// Mitsubishi GX Works2 project: IOCHECK   PLC: Q03UD

PROGRAM MAIN
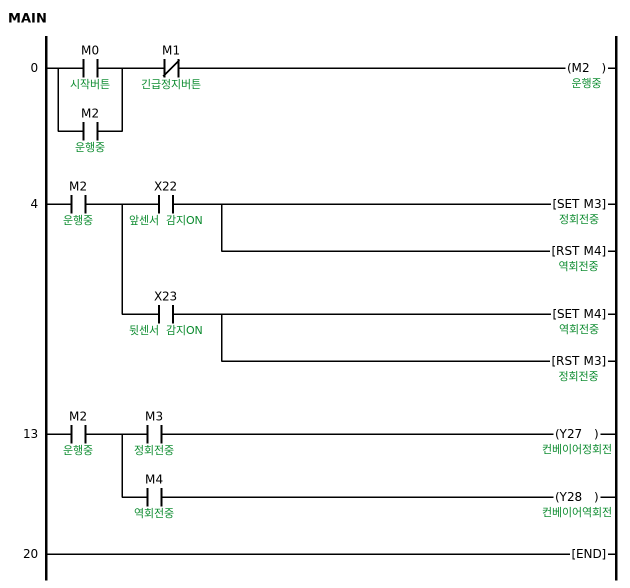
0     LD      M0  ; 시작버튼
      OR      M2  ; 운행중
      ANI     M1  ; 긴급정지버튼
      OUT     M2  ; 운행중
4     LD      M2  ; 운행중
      MPS
      AND     X22  ; 앞센서  감지ON
      SET     M3  ; 정회전중
      RST     M4  ; 역회전중
      MPP
      AND     X23  ; 뒷센서  감지ON
      SET     M4  ; 역회전중
      RST     M3  ; 정회전중
13    LD      M2  ; 운행중
      MPS
      AND     M3  ; 정회전중
      OUT     Y27  ; 컨베이어정회전
      MPP
      AND     M4  ; 역회전중
      OUT     Y28  ; 컨베이어역회전
20    END
END_PROGRAM

PROGRAM IOCHECK
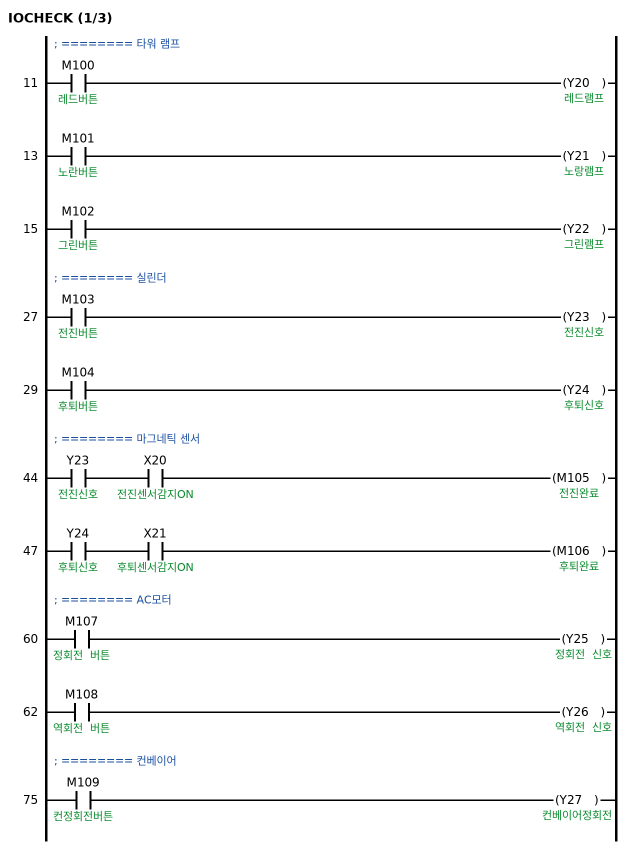
; ======== 타워 램프
11    LD      M100  ; 레드버튼
      OUT     Y20  ; 레드램프
13    LD      M101  ; 노란버튼
      OUT     Y21  ; 노랑램프
15    LD      M102  ; 그린버튼
      OUT     Y22  ; 그린램프
; ======== 실린더
27    LD      M103  ; 전진버튼
      OUT     Y23  ; 전진신호
29    LD      M104  ; 후퇴버튼
      OUT     Y24  ; 후퇴신호
; ======== 마그네틱 센서
44    LD      Y23  ; 전진신호
      AND     X20  ; 전진센서감지ON
      OUT     M105  ; 전진완료
47    LD      Y24  ; 후퇴신호
      AND     X21  ; 후퇴센서감지ON
      OUT     M106  ; 후퇴완료
; ======== AC모터
60    LD      M107  ; 정회전  버튼
      OUT     Y25  ; 정회전  신호
62    LD      M108  ; 역회전  버튼
      OUT     Y26  ; 역회전  신호
; ======== 컨베이어
75    LD      M109  ; 컨정회전버튼
      OUT     Y27  ; 컨베이어정회전
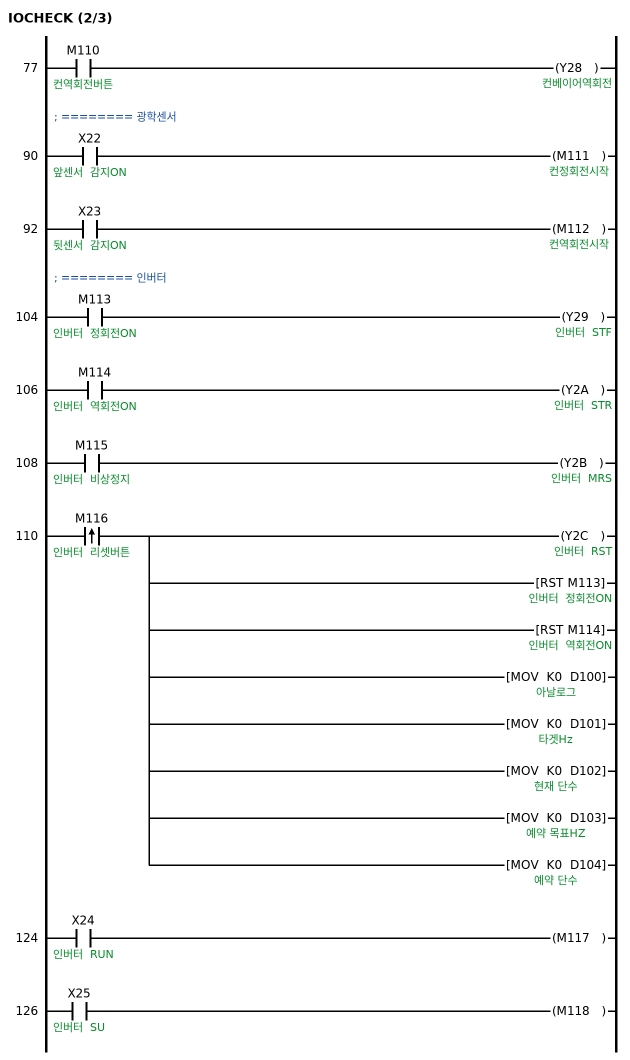
77    LD      M110  ; 컨역회전버튼
      OUT     Y28  ; 컨베이어역회전
; ======== 광학센서
90    LD      X22  ; 앞센서  감지ON
      OUT     M111  ; 컨정회전시작
92    LD      X23  ; 뒷센서  감지ON
      OUT     M112  ; 컨역회전시작
; ======== 인버터
104   LD      M113  ; 인버터  정회전ON
      OUT     Y29  ; 인버터  STF
106   LD      M114  ; 인버터  역회전ON
      OUT     Y2A  ; 인버터  STR
108   LD      M115  ; 인버터  비상정지
      OUT     Y2B  ; 인버터  MRS
110   LDP     M116  ; 인버터  리셋버튼
      OUT     Y2C  ; 인버터  RST
      RST     M113  ; 인버터  정회전ON
      RST     M114  ; 인버터  역회전ON
      MOV     K0 D100  ; 아날로그
      MOV     K0 D101  ; 타겟Hz
      MOV     K0 D102  ; 현재 단수
      MOV     K0 D103  ; 예약 목표HZ
      MOV     K0 D104  ; 예약 단수
124   LD      X24  ; 인버터  RUN
      OUT     M117
126   LD      X25  ; 인버터  SU
      OUT     M118
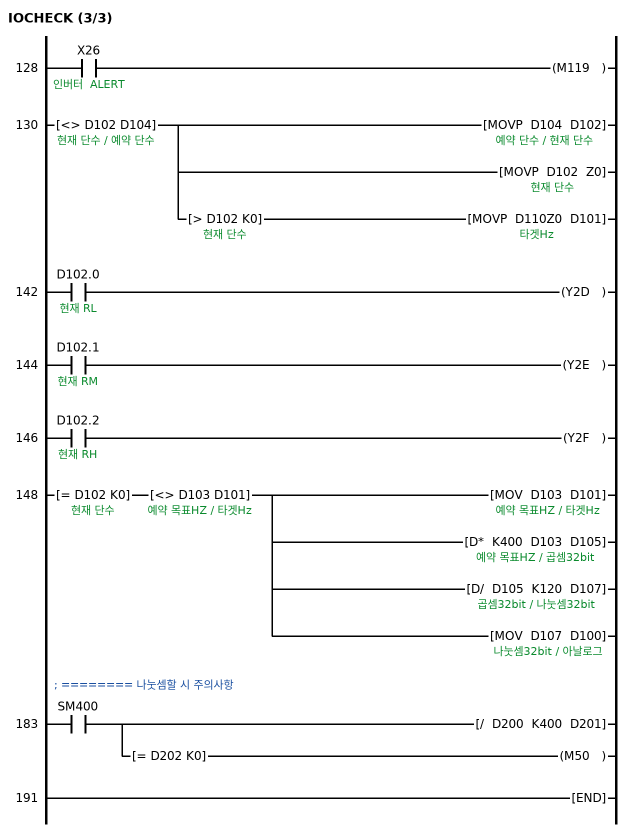
128   LD      X26  ; 인버터  ALERT
      OUT     M119
130   LD<>    D102 D104  ; 현재 단수 / 예약 단수
      MOVP    D104 D102
      MOVP    D102 Z0
      AND>    D102 K0  ; 현재 단수
      MOVP    D110Z0 D101
142   LD      D102.0  ; 현재 RL
      OUT     Y2D
144   LD      D102.1  ; 현재 RM
      OUT     Y2E
146   LD      D102.2  ; 현재 RH
      OUT     Y2F
148   LD=     D102 K0  ; 현재 단수
      AND<>   D103 D101  ; 예약 목표HZ / 타겟Hz
      MOV     D103 D101
      D*      K400 D103 D105  ; 곱셈32bit
      D/      D105 K120 D107  ; 나눗셈32bit
      MOV     D107 D100
; ======== 나눗셈할 시 주의사항
183   LD      SM400
      /       D200 K400 D201
      AND=    D202 K0
      OUT     M50
191   END
END_PROGRAM

PROGRAM INIT
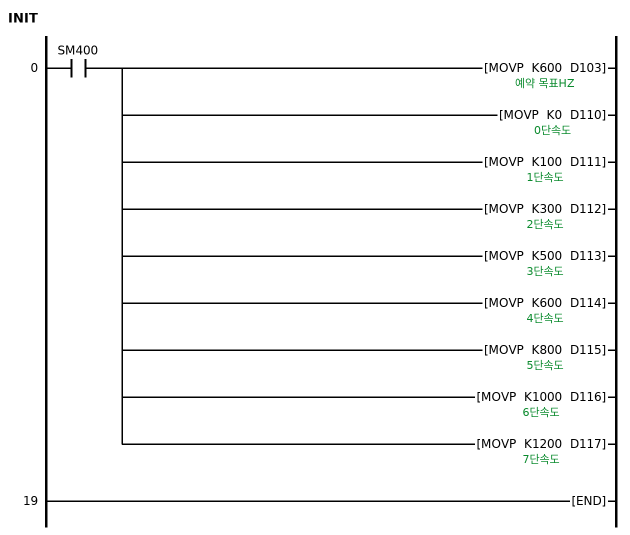
0     LD      SM400
      MOVP    K600 D103  ; 예약 목표HZ
      MOVP    K0 D110  ; 0단속도
      MOVP    K100 D111  ; 1단속도
      MOVP    K300 D112  ; 2단속도
      MOVP    K500 D113  ; 3단속도
      MOVP    K600 D114  ; 4단속도
      MOVP    K800 D115  ; 5단속도
      MOVP    K1000 D116  ; 6단속도
      MOVP    K1200 D117  ; 7단속도
19    END
END_PROGRAM
